FUNCTION F_Laser_Error : FB_Laser
VAR_INPUT
END_VAR
VAR_OUTPUT
	stSetpoints : ST_LaserSetpoints := F_LaserSetpoints();
END_VAR
VAR
	fbLaser : FB_Laser;
END_VAR

fbLaser(
	nVoltageRaw := 0,
	bAmphosOn := TRUE,
	stSetpoints := stSetpoints
);

F_Laser_Error := fbLaser;

END_FUNCTION

(* stored: Version 1.1.0.1, ProductVersion 3.1.4020.14
   POU F_Laser_Error: Id {3fd35628-9ceb-4858-a819-40303a3e6a46}, SpecialFunc None *)
